(* IEC 61131-3 sources: POMIRTS_lab3/AS/Library_2/AsIOLink, 3 files *)

(* ---- AsIOLink.typ ---- *)
TYPE
	ioLinkState_t :
		(
		READY,
		WORK,
		DONE
		);
	ioLinkInternalAccess_t : 	STRUCT  (*internal data*)
		state : ioLinkState_t;
		idCount : UDINT;
		drvInstHandle : UDINT;
		error : UINT;
		done : UDINT;
		serviceResponse : UDINT;
		datatype : USINT;
		buffer : UDINT;
		bufferSize : UDINT;
		bufferFeatures : ARRAY[0..15]OF USINT;
	END_STRUCT;
	ioLinkInternalEvent_t : 	STRUCT  (*internal data*)
		state : ioLinkState_t;
		drvInstHandle : UDINT;
		eventQualifier : USINT;
		eventData : UINT;
		eventLost : BOOL;
		eventPending : BOOL;
		error : UINT;
		bufferFeatures : ARRAY[0..7]OF USINT;
	END_STRUCT;
	ioLinkInternalSetMode_t : 	STRUCT  (*internal data*)
		state : ioLinkState_t;
		error : UINT;
		deviceName : STRING[128];
		channelName : STRING[32];
		accWrite : AsIOAccWrite;
		bufferFeatures : ARRAY[0..7]OF USINT;
	END_STRUCT;
	ioLinkInternalParDownload_t : 	STRUCT  (*internal data*)
		state : ioLinkState_t;
		drvInstHandle : UDINT;
		error : UINT;
		bufferFeatures : ARRAY[0..7]OF USINT;
	END_STRUCT;
END_TYPE

(* ---- AsIOLink.fun ---- *)
{REDUND_CONTEXT} {REDUND_UNREPLICABLE} FUNCTION_BLOCK ioLinkWrite (*write data to an object of the IO-Link device*)
	VAR_INPUT
		enable : BOOL;       (*enables execution*)
		pDeviceName : UDINT; (*device name given as a pointer to string*)
		index : UINT;        (*index to be written*)
		subIndex : USINT;    (*subIndex to be written*)
		datatype : USINT;    (*datatype to be written*)
		pData : UDINT;       (*pointer to the write data*)
		dataLen : UDINT;     (*length of the write access*)
	END_VAR
	VAR_OUTPUT
		errorCode : UINT;   (*error code generated by the IO-Link device*)
		status : UINT;      (*execution status: ERR_OK, ERR_FUB_ENABLE_FALSE, 0xXXXX = see help*)
	END_VAR
	VAR
		_internal : ioLinkInternalAccess_t; (*internal variable*)
	END_VAR
END_FUNCTION_BLOCK

{REDUND_CONTEXT} {REDUND_UNREPLICABLE} FUNCTION_BLOCK ioLinkRead (*read data from an object of the IO-Link device*)
	VAR_INPUT
		enable : BOOL;       (*enables execution*)
		pDeviceName : UDINT; (*device name given as a pointer to string*)
		index : UINT;        (*index to be read*)
		subIndex : USINT;    (*subIndex to be read*)
		datatype : USINT;    (*datatype to be read*)
		pData : UDINT;       (*pointer for the read data*)
		dataLen : UDINT;     (*length of the read data buffer*)
	END_VAR
	VAR_OUTPUT
		errorCode : UINT;    (*error code generated by the IO-Link device*)
		readLen : UDINT;     (*read data size in buffer*)
		status : UINT;       (*execution status: ERR_OK, ERR_FUB_ENABLE_FALSE, 0xXXXX = see help*)
	END_VAR
	VAR
		_internal : ioLinkInternalAccess_t; (*internal variable*)
	END_VAR
END_FUNCTION_BLOCK

{REDUND_CONTEXT} {REDUND_UNREPLICABLE} FUNCTION_BLOCK ioLinkGetEvent (*read event data from event queue*)
	VAR_INPUT
		enable : BOOL;          (*enables execution*)
		pDeviceName : UDINT;    (*device name given as a pointer to string*)
	END_VAR
	VAR_OUTPUT
		eventQualifier : USINT; (*eventQualifier*)
		eventData : UINT;       (*eventData*)
		eventLost : BOOL;       (*is set if some events are overwritten*)
		eventPending : BOOL;    (*indicates if there are more events in the event buffer*)
		status : UINT;          (*execution status: ERR_OK, ERR_FUB_ENABLE_FALSE, 0xXXXX = see help*)
	END_VAR
	VAR
		_internal : ioLinkInternalEvent_t; (*internal variable*)
	END_VAR
END_FUNCTION_BLOCK

{REDUND_CONTEXT} {REDUND_UNREPLICABLE} FUNCTION_BLOCK ioLinkSetMode (*change the mode of an IO-Link device*)
	VAR_INPUT
		enable : BOOL;       (*enables execution*)
		pDeviceName : UDINT; (*device name given as a pointer to string*)
		mode : USINT;        (*desired mode: ioLinkMODE_INACTIVE, ioLinkMODE_DIGINPUT, ioLinkMODE_DIGOUTPUT, ioLinkMODE_FASTOPERATE, ioLinkMODE_OPERATE*)
	END_VAR
	VAR_OUTPUT
		status : UINT;       (*execution status: ERR_OK, ERR_FUB_ENABLE_FALSE, 0xXXXX = see help*)
	END_VAR
	VAR
		_internal : ioLinkInternalSetMode_t; (*internal variable*)
	END_VAR
END_FUNCTION_BLOCK

{REDUND_CONTEXT} {REDUND_UNREPLICABLE} FUNCTION_BLOCK ioLinkParameterDownload (*download the offline configuration to an IO-Link Device*)
	VAR_INPUT
		enable : BOOL;       (*enables execution*)
		pDeviceName : UDINT; (*device name given as a pointer to string*)
	END_VAR
	VAR_OUTPUT
		status : UINT;       (*execution status: ERR_OK, ERR_FUB_ENABLE_FALSE, 0xXXXX = see help*)
	END_VAR
	VAR
		_internal : ioLinkInternalParDownload_t; (*internal variable*)
	END_VAR
END_FUNCTION_BLOCK

(* ---- AsIOLink.var ---- *)
(* error area 37960 - 38009 for AsIOLink reserved *)
VAR CONSTANT
	ioLinkERR_INVALID_PARAMETER : UINT := 37960; (*invalid parameters in function call*)
	ioLinkERR_INVALID_MASTER : UINT := 37961; (*the device is not an IO-Link device or the IO-Link device is not supported *)
	ioLinkERR_COMMUNICATION_DEVICE : UINT := 37962; (*error occured during communication with the IO-Link device e.g. timeout, disconnect, wrong mode ...*)
	ioLinkERR_MAX_OPEN_COUNT : UINT := 37963; (*library client limit is reached*)
	ioLinkERR_REQUESTQUEUE_FULL : UINT := 37964; (*communication request queue if full*)
	ioLinkERR_REQUEST_TO_LONG : UINT := 37965; (*request exceeded allowed length limit*)
	ioLinkERR_BUFFER_TO_SMALL : UINT := 37966; (*device response does not fit in handed receive buffer*)
	ioLinkERR_DEVICE_DRIVER : UINT := 37967; (*error in the ar internal device driver occured*)
	ioLinkERR_DATATYPE_MISMATCH : UINT := 37968; (*the handed datatype length is different to the received data length*)
	ioLinkERR_EVENT_RECEIVED : UINT := 37969; (*an event was received*)
	ioLinkERR_NO_EVENT : UINT := 37970; (*there is no event*)
	ioLinkERR_DEVICE_ERROR : UINT := 37971; (*the IO-Link device returns an error - see errorCode*)
	ioLinkTYPE_SINT : USINT := 2; (*constant for type SINT*)
	ioLinkTYPE_INT : USINT := 3; (*constant for type INT*)
	ioLinkTYPE_DINT : USINT := 4; (*constant for type DINT*)
	ioLinkTYPE_LINT : USINT := 23; (*constant for type LINT*)
	ioLinkTYPE_USINT : USINT := 5; (*constant for type USINT*)
	ioLinkTYPE_UINT : USINT := 6; (*constant for type UINT*)
	ioLinkTYPE_UDINT : USINT := 7; (*constant for type UDINT*)
	ioLinkTYPE_ULINT : USINT := 10; (*constant for type ULINT*)
	ioLinkTYPE_REAL : USINT := 8; (*constant for type REAL*)
	ioLinkTYPE_LREAL : USINT := 14; (*constant for type LREAL*)
	ioLinkTYPE_STRING : USINT := 9; (*constant for type STRING*)
	ioLinkTYPE_RECORD : USINT := 254; (*constant for type RECORD*)
	ioLinkMODE_INACTIVE : USINT := 0; (*constant for operating mode digital output*)
	ioLinkMODE_DIGINPUT : USINT := 1; (*constant for operating mode digital input*)
	ioLinkMODE_DIGOUTPUT : USINT := 2; (*constant for operating mode digital output*)
	ioLinkMODE_OPERATE : USINT := 10; (*constant for operating mode operate*)
END_VAR
